// TIA Portal V20 export
TYPE "OPC_DsetRequest"
// stored: Namespace ProductionLine
   STRUCT
      SourceSeq : Int;   // // Communication flag, described in the Request - Response tab
      DecisionPoint : String[30];   // // Machine/workstation code: - DP1,…, DP4
      Barcode : String[30];   // // Unique identification of scanned KLTs. For NoRead use ??????????
   END_STRUCT;
END_TYPE
